// Owner-local recipe engineering data: model identities and their typed Unit records.
// Generic validation/storage remains in FB_LocalRecipeProvider; process behavior
// remains in the project-owned FB_PressDemoUnit. MAIN only composes the two.
FUNCTION_BLOCK FB_PressRecipeCatalog
VAR_OUTPUT
    {attribute 'OPC.UA.DA' := '0'}
    Provider : FB_LocalRecipeProvider;
END_VAR
VAR PERSISTENT
    // §3.8b - the records are edited through the Unit (the active model's PAR_CFG)
    // and must outlive a restart, so they are retained and seeded only once.
    _default : ST_PneumaticPressParCfg;
    _aluminum : ST_PneumaticPressParCfg;
    _plastic : ST_PneumaticPressParCfg;
    _steel : ST_PneumaticPressParCfg;
    _seeded : UINT;               // RECIPE_SEED once the defaults below were written
END_VAR
VAR
    _model : ST_ModelId;
    _configured : BOOL;
END_VAR
VAR CONSTANT
    // Bump to re-seed every record with the design values below (a download that
    // changes them, or a record layout change).
    RECIPE_SEED : UINT := 1;
END_VAR

// Static catalog: no cyclic work.

METHOD Setup : BOOL
VAR_INPUT
    UnitRef : REFERENCE TO FB_PressDemoUnit;
END_VAR
VAR
    Ok : BOOL;
END_VAR
IF _configured THEN
    Setup := TRUE;
    RETURN;
END_IF

// §8.11 per-model performance references: IdealCycleMs feeds OEE Performance
// (§8.5.1); BaselineWorkMs arms the WORK-time degradation watch (§8.11.4(d)).
// Values = design cycle for this training cell (motions + settle + dwell).
// Seeded once: afterwards the retained records hold what was edited.
IF _seeded <> RECIPE_SEED THEN
    _default.PressSettleTime := T#500MS;
    _default.TransferSettleTime := T#100MS;
    _default.IdealCycleMs := 6000;
    _default.BaselineWorkMs := 6000;
    _aluminum.PressSettleTime := T#300MS;
    _aluminum.TransferSettleTime := T#80MS;
    _aluminum.IdealCycleMs := 5700;
    _aluminum.BaselineWorkMs := 5700;
    _plastic.PressSettleTime := T#650MS;
    _plastic.TransferSettleTime := T#120MS;
    _plastic.IdealCycleMs := 6200;
    _plastic.BaselineWorkMs := 6200;
    _steel.PressSettleTime := T#1200MS;
    _steel.TransferSettleTime := T#150MS;
    _steel.IdealCycleMs := 6800;
    _steel.BaselineWorkMs := 6800;
    _seeded := RECIPE_SEED;
END_IF

Ok := Provider.Register(ModelCode := '', RecipeKey := 'PneumaticPressUnit',
    pData := ADR(_default), Size := SIZEOF(_default));
Ok := Provider.Register(ModelCode := 'ALUMINUM', RecipeKey := 'PneumaticPressUnit',
    pData := ADR(_aluminum), Size := SIZEOF(_aluminum)) AND Ok;
Ok := Provider.Register(ModelCode := 'PLASTIC', RecipeKey := 'PneumaticPressUnit',
    pData := ADR(_plastic), Size := SIZEOF(_plastic)) AND Ok;
Ok := Provider.Register(ModelCode := 'STEEL', RecipeKey := 'PneumaticPressUnit',
    pData := ADR(_steel), Size := SIZEOF(_steel)) AND Ok;

_model.ModelCode := 'ALUMINUM';
Ok := UnitRef.RegisterAvailableModel(Id := _model) AND Ok;
_model.ModelCode := 'PLASTIC';
Ok := UnitRef.RegisterAvailableModel(Id := _model) AND Ok;
_model.ModelCode := 'STEEL';
Ok := UnitRef.RegisterAvailableModel(Id := _model) AND Ok;
Ok := UnitRef.SetRecipeCatalog(pCatalog := THIS) AND Ok;

_configured := Ok;
Setup := Ok;
END_METHOD

// §3.8a - write an edited recipe back to the record of its model, so the next
// changeover to that model loads it. FALSE for a model this catalog does not hold.
METHOD M_Store : BOOL
VAR_INPUT
    ModelCode : STRING(64);
    Record    : ST_PneumaticPressParCfg;
END_VAR
M_Store := TRUE;
IF ModelCode = '' THEN
    _default := Record;
ELSIF ModelCode = 'ALUMINUM' THEN
    _aluminum := Record;
ELSIF ModelCode = 'PLASTIC' THEN
    _plastic := Record;
ELSIF ModelCode = 'STEEL' THEN
    _steel := Record;
ELSE
    M_Store := FALSE;
END_IF
END_METHOD

END_FUNCTION_BLOCK

(* stored: Version 1.1.0.1, ProductVersion 3.1.4024.12
   POU FB_PressRecipeCatalog: Id {f1bc98f5-6ad1-4105-bbca-cdb707f304e6}, SpecialFunc None
   Method Setup: Id {f3703336-44cb-4ed4-a15f-6dc17b858973}
   Method M_Store: Id {5f8f75d4-bd85-4c3d-a0f4-7f6f85b97e42} *)
